FUNCTION TFCoppiaPinzaOk : BOOL // True
VAR_INPUT
	Coppia_Attuale : REAL;	// Coppia attuale asse
	Coppia_Riferimento : REAL; // Coppia che si desidera che sia presente
	Offset_Controllo : REAL; // Valore che determina la finestra di controllo rispetto al valore di riferimento
END_VAR
VAR
END_VAR


TFCoppiaPinzaOk := FALSE;
				
IF (ABS(Coppia_Attuale) >= Coppia_Riferimento - Offset_Controllo AND (ABS(Coppia_Attuale) <= Coppia_Riferimento + Offset_Controllo)) THEN
	TFCoppiaPinzaOk := TRUE;
	RETURN;
END_IF

END_FUNCTION

(* stored: Version 1.1.0.1, ProductVersion 3.1.4024.11
   POU TFCoppiaPinzaOk: Id {d76eeba9-88fd-4924-be98-1a5d510a22d0}, SpecialFunc None *)
